# EPICS substitutions: bk1787b/bk1787bApp/Db/bk_1787b.substitutions
file bk_1787b.template { pattern
{ Sys	, Dev		,PORT		}
{ Depo	, "{BK:PS}"	, Depo_PS2	}
}
